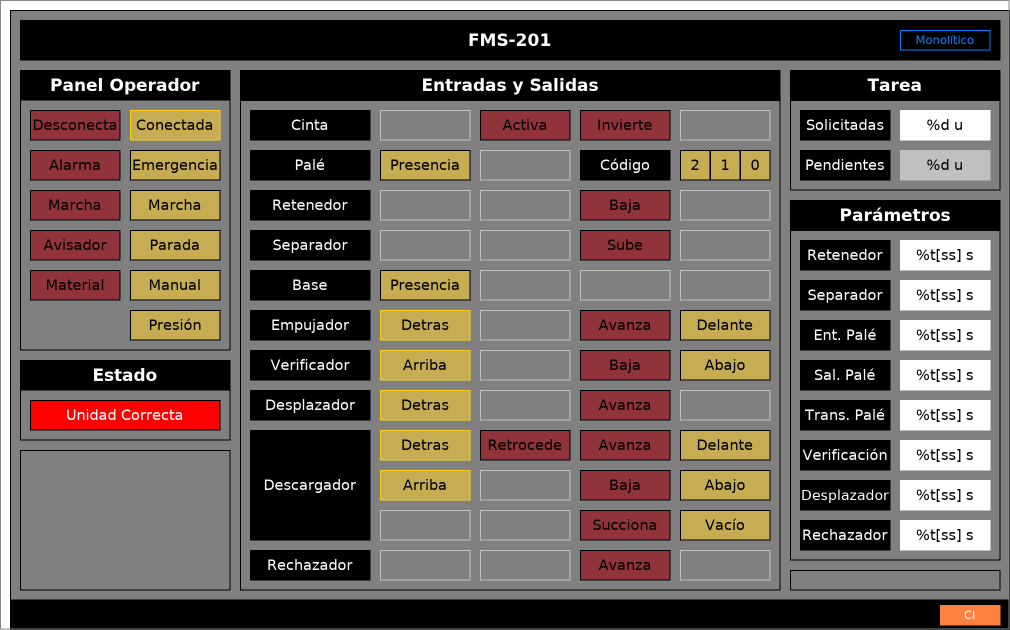
VISUALIZATION V_Estacion  // 1010x630
    Rectangle (10,10 1000x590)
    Rectangle (240,100 540x490)
    Rectangle (20,70 210x280)
    Rectangle (30,110 90x30), "Desconecta"
        tap MAIN.Estacion.o_DesconectaEstacion
    Rectangle (30,150 90x30), "Alarma"
        toggle MAIN.Estacion.o_LamparaAlarma
    Rectangle (30,190 90x30), "Marcha"
        toggle MAIN.Estacion.o_LamparaMarcha
    Rectangle (30,230 90x30), "Avisador"
        tap MAIN.Estacion.o_AvisadorSonoro
    Rectangle (30,270 90x30), "Material"
        toggle MAIN.Estacion.o_LamparaMaterial
    Rectangle (130,110 90x30), "Conectada"
        toggle MAIN.Estacion.i_EstacionConectada
    Rectangle (130,150 90x30), "Emergencia"
        toggle MAIN.Estacion.i_PulsadorEmergencia
    Rectangle (130,190 90x30), "Marcha"
        tap MAIN.Estacion.i_PulsadorMarcha
    Rectangle (130,230 90x30), "Parada"
        tap MAIN.Estacion.i_PulsadorParada p1329445385=TRUE
    Rectangle (130,270 90x30), "Manual"
        toggle MAIN.Estacion.i_SelectorManual
    Rectangle (20,70 210x30), "Panel Operador"
    Rectangle (240,70 540x30), "Entradas y Salidas"
    Rectangle (250,110 120x30), "Cinta"
    Rectangle (250,150 120x30), "Palé"
    Rectangle (250,190 120x30), "Retenedor"
    Rectangle (250,230 120x30), "Separador"
    Rectangle (250,430 120x110), "Descargador"
    Rectangle (250,550 120x30), "Rechazador"
    Rectangle (250,350 120x30), "Verificador"
    Rectangle (250,390 120x30), "Desplazador"
    Rectangle (250,310 120x30), "Empujador"
    Rectangle (480,110 90x30), "Activa"
        toggle MAIN.Estacion.o_CintaActiva
    Rectangle (380,110 90x30)
    Rectangle (580,110 90x30), "Invierte"
        toggle MAIN.Estacion.o_CintaInvierte
    Rectangle (680,110 90x30)
    Rectangle (380,150 90x30), "Presencia"
        toggle MAIN.Estacion.i_PresenciaPale
    Rectangle (480,150 90x30)
    Rectangle (580,150 90x30), "Código"
    Rectangle (680,150 30x30), "2"
        toggle MAIN.Estacion.i_CodigoPaleBit2
    Rectangle (710,150 30x30), "1"
        toggle MAIN.Estacion.i_CodigoPaleBit1
    Rectangle (740,150 30x30), "0"
        toggle MAIN.Estacion.i_CodigoPaleBit0
    Rectangle (380,190 90x30)
    Rectangle (580,190 90x30), "Baja"
        toggle MAIN.Estacion.o_RetenedorBaja
    Rectangle (680,190 90x30)
    Rectangle (480,230 90x30)
    Rectangle (580,230 90x30), "Sube"
        toggle MAIN.Estacion.o_SeparadorSube
    Rectangle (380,230 90x30)
    Rectangle (680,230 90x30)
    Rectangle (580,310 90x30), "Avanza"
        toggle MAIN.Estacion.o_EmpujadorAvanza
    Rectangle (380,310 90x30), "Detras"
        toggle MAIN.Estacion.i_EmpujadorDetras
    Rectangle (480,310 90x30)
    Rectangle (580,350 90x30), "Baja"
        toggle MAIN.Estacion.o_VerificardorBaja
    Rectangle (480,350 90x30)
    Rectangle (580,390 90x30), "Avanza"
        toggle MAIN.Estacion.o_DesplazadorAvanza
    Rectangle (580,430 90x30), "Avanza"
        toggle MAIN.Estacion.o_DescargadorAvanza
    Rectangle (480,430 90x30), "Retrocede"
        toggle MAIN.Estacion.o_DescargadorRetrocede
    Rectangle (480,190 90x30)
    Rectangle (580,470 90x30), "Baja"
        toggle MAIN.Estacion.o_DescargadorBaja
    Rectangle (580,510 90x30), "Succiona"
        toggle MAIN.Estacion.o_DescargadorSucciona
    Rectangle (580,550 90x30), "Avanza"
        toggle MAIN.Estacion.o_RechazadorAvanza
    Rectangle (480,550 90x30)
    Rectangle (480,390 90x30)
    Rectangle (480,470 90x30)
    Rectangle (480,510 90x30)
    Rectangle (680,310 90x30), "Delante"
        toggle MAIN.Estacion.i_EmpujadorDelante
    Rectangle (380,350 90x30), "Arriba"
        toggle MAIN.Estacion.i_VerificadorArriba
    Rectangle (680,350 90x30), "Abajo"
        toggle MAIN.Estacion.i_VerificadorAbajo
    Rectangle (380,390 90x30), "Detras"
        toggle MAIN.Estacion.i_DesplazadorDetras
    Rectangle (680,390 90x30)
    Rectangle (680,550 90x30)
    Rectangle (380,550 90x30)
    Rectangle (380,510 90x30)
    Rectangle (380,430 90x30), "Detras"
        toggle MAIN.Estacion.i_DescargadorDetras
    Rectangle (680,430 90x30), "Delante"
        toggle MAIN.Estacion.i_DescargadorDelante
    Rectangle (380,470 90x30), "Arriba"
        toggle MAIN.Estacion.i_DescargadorArriba
    Rectangle (680,470 90x30), "Abajo"
        toggle MAIN.Estacion.i_DescargadorAbajo
    Rectangle (680,510 90x30), "Vacío"
        toggle MAIN.Estacion.i_DescargadorVacio
    Rectangle (20,20 980x40), "FMS-201"
    Rectangle (20,360 210x80)
    Rectangle (900,30 90x20), "Monolítico"
    Rectangle (130,310 90x30), "Presión"
        toggle MAIN.Estacion.i_DetectorPresion
    Rectangle (10,600 1000x30)
    Rectangle (940,605 60x20), "CI", colour toggle: MAIN.Estacion.CondicionInicial
    Rectangle (790,100 210x90)
    Rectangle (790,70 210x30), "Tarea"
    Rectangle (790,230 210x330)
    Rectangle (790,200 210x30), "Parámetros"
    Rectangle (800,320 90x30), "Ent. Palé"
    Rectangle (900,320 90x30), "%t[ss] s", text variable: MAIN.Estacion.TiempoEntradaPale
        OnMouseClick: write the text variable via Default
    Rectangle (800,440 90x30), "Verificación"
    Rectangle (900,440 90x30), "%t[ss] s", text variable: MAIN.Estacion.TiempoVerificacion
        OnMouseClick: write the text variable via Default
    Rectangle (800,480 90x30), "Desplazador"
    Rectangle (900,480 90x30), "%t[ss] s", text variable: MAIN.Estacion.TiempoDesplazador
        OnMouseClick: write the text variable via Default
    Rectangle (800,520 90x30), "Rechazador"
    Rectangle (900,520 90x30), "%t[ss] s", text variable: MAIN.Estacion.TiempoRechazador
        OnMouseClick: write the text variable via Default
    Rectangle (800,360 90x30), "Sal. Palé"
    Rectangle (900,360 90x30), "%t[ss] s", text variable: MAIN.Estacion.TiempoEntradaPale
        OnMouseClick: write the text variable via Default
    Rectangle (800,400 90x30), "Trans. Palé"
    Rectangle (900,400 90x30), "%t[ss] s", text variable: MAIN.Estacion.TiempoEntradaPale
        OnMouseClick: write the text variable via Default
    Rectangle (30,400 190x30), "Unidad Correcta", colour toggle: MAIN.Estacion.UnidadCorrecta
    Rectangle (800,110 90x30), "Solicitadas"
    Rectangle (800,150 90x30), "Pendientes"
    Rectangle (900,110 90x30), "%d u", text variable: MAIN.Estacion.UnidadesSolicitadas
        OnMouseClick: write the text variable via Default
    Rectangle (900,150 90x30), "%d u", text variable: MAIN.Estacion.UnidadesPendientes
    Rectangle (250,270 120x30), "Base"
    Rectangle (380,270 90x30), "Presencia"
        toggle MAIN.Estacion.i_PresenciaBase
    Rectangle (480,270 90x30)
    Rectangle (680,270 90x30)
    Rectangle (580,270 90x30)
    Rectangle (800,240 90x30), "Retenedor"
    Rectangle (900,240 90x30), "%t[ss] s", text variable: MAIN.Estacion.TiempoRetenedor
        OnMouseClick: write the text variable via Default
    Rectangle (800,280 90x30), "Separador"
    Rectangle (900,280 90x30), "%t[ss] s", text variable: MAIN.Estacion.TiempoSeparador
        OnMouseClick: write the text variable via Default
    Rectangle (20,360 210x30), "Estado"
    Rectangle (20,450 210x140)
    Rectangle (790,570 210x20)
END_VISUALIZATION

(* stored: Version 1.1.0.1
   Visu V_Estacion: Id {9af79785-e2fb-4053-b627-6176b8bb155f} *)
